// TIA Portal project "babu_2Switch2ValvePriority" (V15)

(* hardware
DEVICE "S7-1200 station_1"  S7-1200 Station
   slot 0: "Rack_0"  S7-1200 Rack  Rack  V1.0
   slot 1: "PLC_1"  CPU 1212C DC/DC/DC  6ES7 212-1AE40-0XB0  V4.2
*)

// ===== PLC "PLC_1"  CPU 1212C DC/DC/DC =====

VAR_GLOBAL   // PLC tag table "Default tag table"
   "S1" AT %M0.0 : Bool;
   "VALVE 1" AT %Q0.0 : Bool;
   "VALVE 2" AT %Q0.1 : Bool;
   "S2" AT %M0.1 : Bool;
   "MEMORY" AT %M0.2 : Bool;
   "PRIORITY OVERRIDE" AT %Q0.2 : Bool;
END_VAR

ORGANIZATION_BLOCK "Main"   // OB1, LAD, ProgramCycle
TITLE = "Main Program Sweep (Cycle)"
{ S7_Optimized_Access := 'TRUE' }
VERSION : 0.1
   VAR_INPUT
      Initial_Call : Bool;   // Initial call of this OB
      Remanence : Bool;   // =True, if remanent data are available
   END_VAR
BEGIN

REGION Network 1
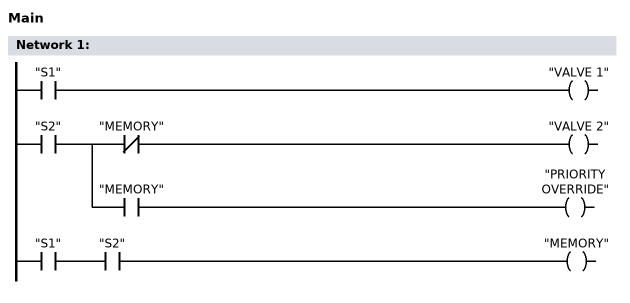
   RUNG wire#powerrail
      Contact( "S1" )
      Coil( "VALVE 1" )
   END_RUNG
   RUNG wire#powerrail
      Contact( "S2" )
      wire#w1
      I_Contact( "MEMORY" )
      Coil( "VALVE 2" )
   END_RUNG
   RUNG wire#w1
      Contact( "MEMORY" )
      Coil( "PRIORITY OVERRIDE" )
   END_RUNG
   RUNG wire#powerrail
      Contact( "S1" )
      Contact( "S2" )
      Coil( "MEMORY" )
   END_RUNG
   // the same network as SCL:
   "VALVE 1" := "S1";
   "VALVE 2" := "S2" AND NOT "MEMORY";
   "PRIORITY OVERRIDE" := "S2" AND "MEMORY";
   "MEMORY" := "S1" AND "S2";
END_REGION
END_ORGANIZATION_BLOCK